PROGRAM Reaktoreinheit
VAR
	// Allgemeine Instanziierungen
	Mode					:FB_Modus;
	
	// Instanziierung der Sensoren
	T1						:FB_S_Sensor;
	F1						:FB_S_Sensor;
	// Instanziierung der Aktoren
	YSE1, YSE2				:FB_A_Magnetventil;
	YSA1, YSA2, YSA3		:FB_A_Magnetventil;
	YSP1, YSP2, YSP3		:FB_A_Magnetventil;
	
	NC1						:FB_A_Motor1R;
	
	PS1						:FB_A_Motor2R;
	
	HKP1					:FB_A_HKSystem;
END_VAR

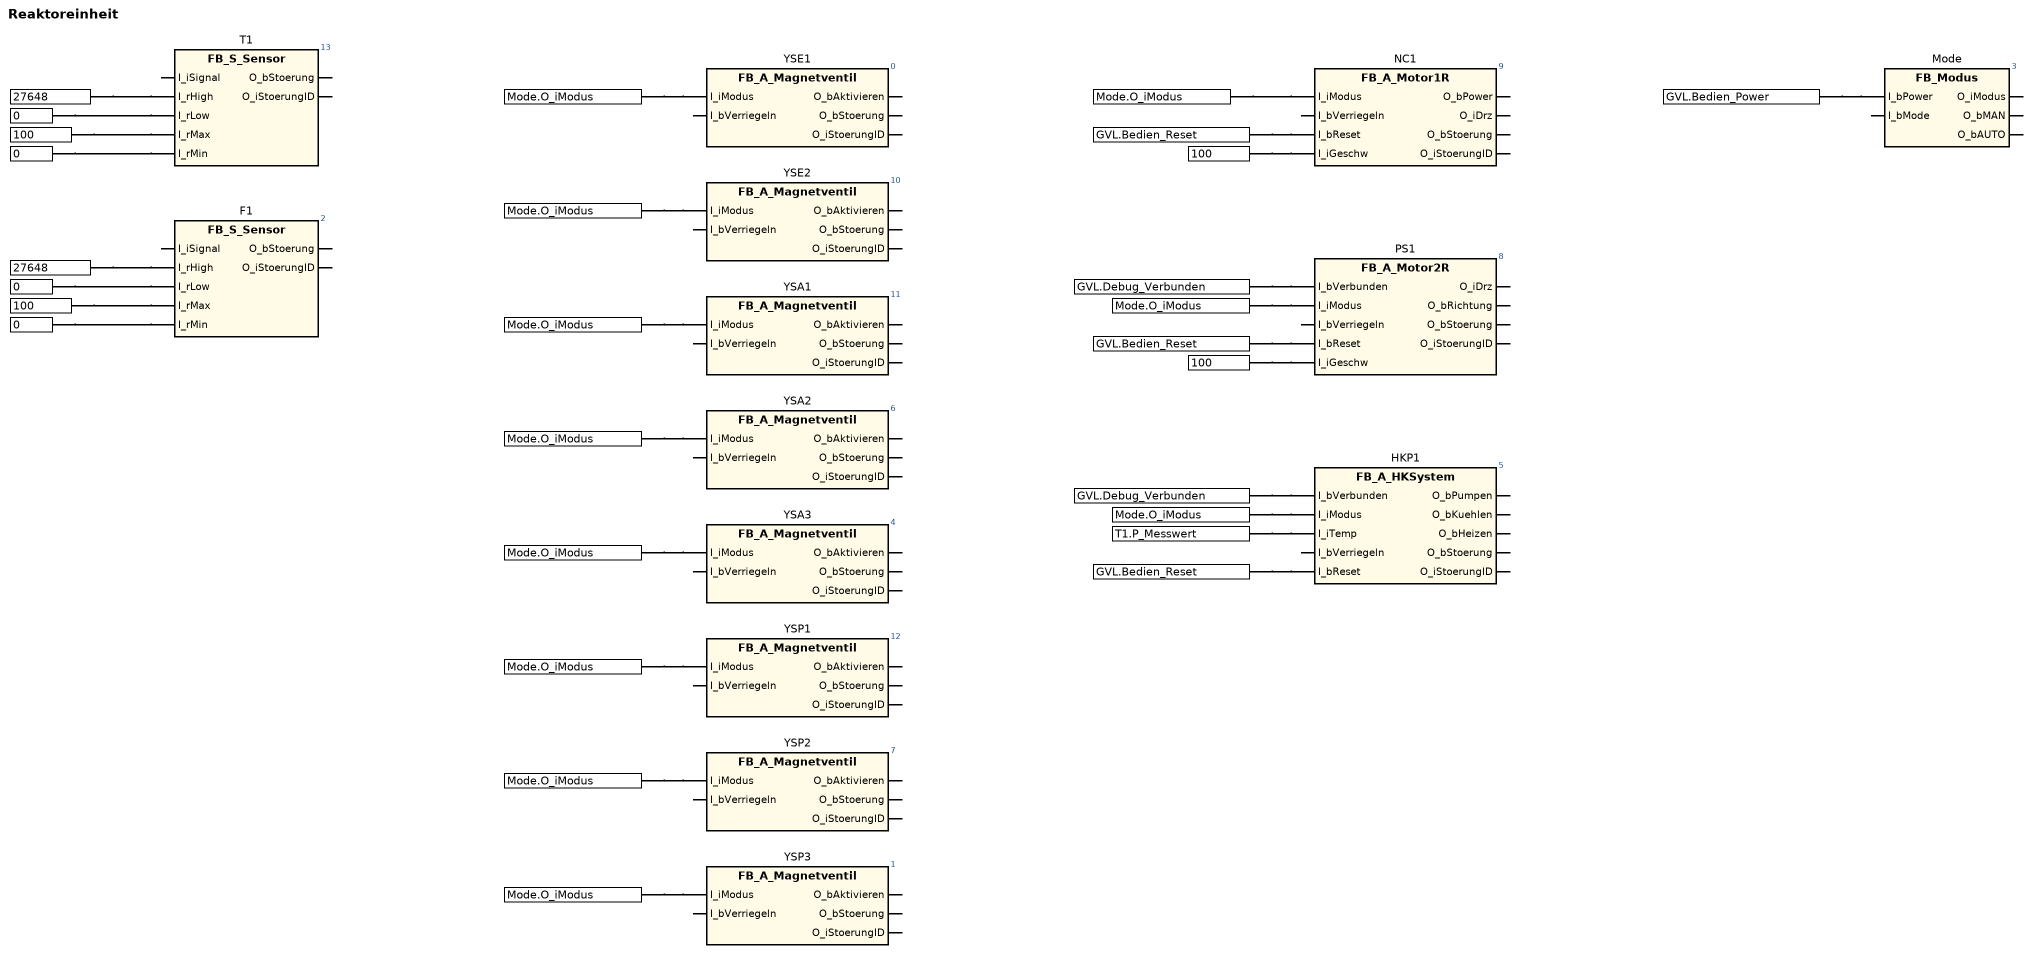
YSE1(I_iModus := Mode.O_iModus); // FB_A_Magnetventil
YSP3(I_iModus := Mode.O_iModus); // FB_A_Magnetventil
F1(I_rHigh := 27648, I_rLow := 0, I_rMax := 100, I_rMin := 0); // FB_S_Sensor
Mode(I_bPower := GVL.Bedien_Power); // FB_Modus
YSA3(I_iModus := Mode.O_iModus); // FB_A_Magnetventil
HKP1(
    I_bVerbunden := GVL.Debug_Verbunden,
    I_iModus := Mode.O_iModus,
    I_iTemp := T1.P_Messwert,
    I_bReset := GVL.Bedien_Reset); // FB_A_HKSystem
YSA2(I_iModus := Mode.O_iModus); // FB_A_Magnetventil
YSP2(I_iModus := Mode.O_iModus); // FB_A_Magnetventil
PS1(
    I_bVerbunden := GVL.Debug_Verbunden,
    I_iModus := Mode.O_iModus,
    I_bReset := GVL.Bedien_Reset,
    I_iGeschw := 100); // FB_A_Motor2R
NC1(I_iModus := Mode.O_iModus, I_bReset := GVL.Bedien_Reset, I_iGeschw := 100); // FB_A_Motor1R
YSE2(I_iModus := Mode.O_iModus); // FB_A_Magnetventil
YSA1(I_iModus := Mode.O_iModus); // FB_A_Magnetventil
YSP1(I_iModus := Mode.O_iModus); // FB_A_Magnetventil
T1(I_rHigh := 27648, I_rLow := 0, I_rMax := 100, I_rMin := 0); // FB_S_Sensor

END_PROGRAM

(* stored: Version 1.1.0.1, ProductVersion 3.1.4024.12
   POU Reaktoreinheit: Id {cd9b3003-448b-4d1c-90df-494b3fb1e47a}, SpecialFunc None *)
